// TIA Portal V18 export
TYPE "UDT_AHUsRegulatorsDataType"
// stored: IsFailsafeCompliant false
   STRUCT
      cTempCooling : Array[1..3] of Byte;
      cTempHeating : Array[1..3] of Byte;
      cIAQ : Array[1..3] of Byte;
      cBuildingdP : Array[1..3] of Byte;
   END_STRUCT;
END_TYPE
